// TIA Portal V20 export
DATA_BLOCK "HmiInterface"   // DB41
// stored: Access Published, MemoryReserve 100, Namespace Unit1.Em6
   VAR
      em : "LAF_typeEmInterface";
      hotPressLeft { S7_SetPoint := 'True'} : "LER_typeSequenceInterface";
      cmHotpressLeftSafetyPin : "LBC_typeDigitalSignalInterface";
      cmHotpressLeftJRDetect : "LBC_typeDigitalSignalInterface";
      cmHotpressLeftStageLiftFrontUpDown : "LBC_typeTwoWayActuatorInterface";
      cmHotpressLeftStageLiftRearUpDown : "LBC_typeTwoWayActuatorInterface";
      cmHotpressLeftStageLiftAllUpDown : "LBC_typeTwoWayActuatorInterface";
      cmHotPressLeftServoPress : "LER_typeServoPressInterface";
      cmHotPressLeftTemperature : "LER_typeHeaterInterface";
   END_VAR
   VAR RETAIN
      cmHotPressLeftHistory : "LER_typeServoPressHistory";
   END_VAR
   VAR
      intCondition : "Unit1.Em6.typeIntConditionHmiInterface";
   END_VAR
BEGIN
   cmHotPressLeftTemperature.configuration.E5CC[2..5].Temp_SP := 0;
   cmHotPressLeftTemperature.configuration.E5CC[2..5].Temp_AlarmValue1 := 0;
   cmHotPressLeftTemperature.configuration.E5CC[1..5].Temp_AlarmValue1_UpperLimit := 45;
   cmHotPressLeftTemperature.configuration.E5CC[1..5].Temp_AlarmValue1_LowerLimit := 15;
   cmHotPressLeftTemperature.configuration.E5CC[2..5].Temp_AlarmValue2 := 0;
   cmHotPressLeftTemperature.configuration.E5CC[1..5].Temp_AlarmValue2_UpperLimit := 42;
   cmHotPressLeftTemperature.configuration.E5CC[1..5].Temp_AlarmValue2_LowerLimit := 18;
   cmHotPressLeftTemperature.configuration.E5CC[1..5].Temp_Upper_Limit_Temp := 40;
   cmHotPressLeftTemperature.configuration.E5CC[1..5].Temp_Lower_Limit_Temp := 20;
   cmHotPressLeftTemperature.configuration.E5CC[2..5].Temp_MC_Off_Value := 0;
   cmHotPressLeftTemperature.configuration.E5CC[1..5].Temp_Upper_Complete_Range := 1;
   cmHotPressLeftTemperature.configuration.E5CC[1..5].Temp_Lower_Complete_Range := -1;
END_DATA_BLOCK
